FUNCTION_BLOCK SupplyConv (* Composite Function Block Type *)
  (* Standard: 61499-2 *)
  (* Version 1.0, 2020-03-21, Duc Do Tran, OFFIS e.V. *)
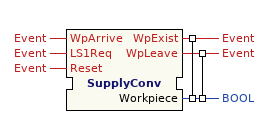
  EVENT_INPUT
    WpArrive; (* Normal Execution Request *)
    LS1Req;
    Reset;
  END_EVENT
  EVENT_OUTPUT
    WpExist WITH Workpiece; (* Execution Confirmation *)
    WpLeave WITH Workpiece;
  END_EVENT
  VAR_OUTPUT
    Workpiece : BOOL; (* Output event qualifier *)
  END_VAR
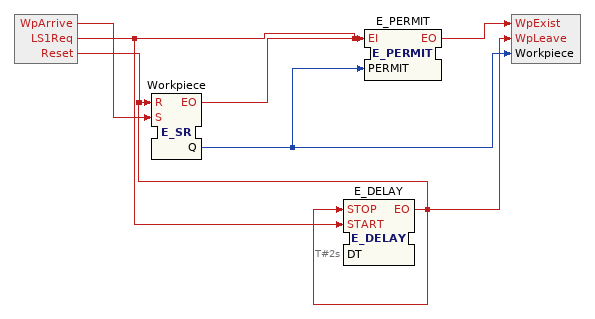
  FBS
    E_DELAY : E_DELAY(DT := T#2s);
    E_PERMIT : E_PERMIT;
    Workpiece : E_SR;
  END_FBS
  EVENT_CONNECTIONS
    E_DELAY.EO TO Workpiece.R;
    E_DELAY.EO TO E_DELAY.STOP;
    Workpiece.EO TO E_PERMIT.EI;
    WpArrive TO Workpiece.S;
    E_PERMIT.EO TO WpExist;
    E_DELAY.EO TO WpLeave;
    LS1Req TO E_DELAY.START;
    LS1Req TO E_PERMIT.EI;
    Reset TO Workpiece.R;
  END_CONNECTIONS
  DATA_CONNECTIONS
    Workpiece.Q TO E_PERMIT.PERMIT;
    Workpiece.Q TO Workpiece;
  END_CONNECTIONS
END_FUNCTION_BLOCK
